Staubli VAL3: CartesianVel.dtx

public num resVel
public num cv[6]
